// TIA Portal V20 export
DATA_BLOCK "DB_ChillerSMC"   // DB541
// stored: AutoNumber false, InstanceOfName FB_ChillerSMC, InstanceOfType FB
"FB_ChillerSMC"
   // VAR
   //    sTimeHeadChillerCutOff { S7_SetPoint := 'True'} : TON_TIME;
   //    sTimeHeadChillerTemperature { S7_SetPoint := 'True'} : TON_TIME;
   //    sTimeSourceChillerCutOff { S7_SetPoint := 'True'} : TON_TIME;
   //    sTimeSourceChillerTemperature { S7_SetPoint := 'True'} : TON_TIME;
   // END_VAR
BEGIN
END_DATA_BLOCK
